(* IEC 61131-3 sources: Std_PalletMover/Class/HAL_BMS_Base, 1 file *)

(* ---- HAL_BMS_Base.st ---- *)
#define COMM_TIMEOUT              1000    // ms before timeout
#define TIMEOUTDELAY              15000    // Delay before checking for a communication timeout.

(*!
<Class
	Name               = "HAL_BMS_Base"
	Revision           = "0.0"
	RealtimeTask       = "false"
	CyclicTask         = "false"
	BackgroundTask     = "false"
	Sigmatek           = "false"
	OSInterface        = "false"
	HighPriority       = "false"
	Automatic          = "false"
	UpdateMode         = "Prescan"
	SharedCommandTable = "true"
	Objectsize         = "(284,120)">
	<Channels>
		<Server Name="ClassSvr" Visualized="false" Initialize="false" WriteProtected="true" Retentive="false"/>
	</Channels>
</Class>
*)
HAL_BMS_Base : CLASS
	TYPE
	  tBMSAlarms : BDINT  //! <Type Public="true" Name="tBMSAlarms"/>
	  [
	    1 ba_OverVoltage,
	    2 ba_UnderVoltage,
	    3 ba_AlmostUnderVoltage,
	    4 ba_BatteryEmpty,
	    5 ba_BatteryAlmostEmpty,
	    6 ba_InternalDefect,
	    7 ba_NoCommunication,
	    8 Bit8,
	    9 Bit9,
	    10 Bit10,
	    11 Bit11,
	    12 Bit12,
	    13 Bit13,
	    14 Bit14,
	    15 Bit15,
	    16 Bit16,
	    17 Bit17,
	    18 Bit18,
	    19 Bit19,
	    20 Bit20,
	    21 Bit21,
	    22 Bit22,
	    23 Bit23,
	    24 Bit24,
	    25 Bit25,
	    26 Bit26,
	    27 Bit27,
	    28 Bit28,
	    29 Bit29,
	    30 Bit30,
	    31 Bit31,
	    32 Bit32,
	  ];
#pragma pack(push, 1)
	  tBMSData : STRUCT  //! <Type Public="true" Name="tBMSData"/>
	    bd_StateOfCharge : UINT;
	    bd_TimeToGo : UINT;
	    bd_EnergyDraw : INT;
	    bd_BatteryVoltage : UINT;
	    bd_BatteryCurrent : INT;
	    bd_BatteryTemperature : INT;
	    bd_BatteryCharging : BOOL;
	    bd_BatteryLowIndication : BOOL;
	    bd_Alarm : tBMSAlarms;
	  END_STRUCT;
#pragma pack(pop)
	END_TYPE
  //Servers:
	ClassSvr 	: SvrChCmd_DINT;
  //Clients:
  //Variables:
  //Functions:

	FUNCTION VIRTUAL GLOBAL GetBMSData
		VAR_OUTPUT
			returnValue 	: tBMSData;
		END_VAR;
  //Tables:
	FUNCTION @STD
		VAR_OUTPUT
			ret_code	: CONFSTATES;
		END_VAR;
	FUNCTION GLOBAL TAB @CT_;
END_CLASS;

FUNCTION VIRTUAL GLOBAL HAL_BMS_Base::GetBMSData
  #pragma warning(disable: 73);
  #pragma warning(disable: 76);
	VAR_OUTPUT
		returnValue 	: tBMSData;
	END_VAR
  #pragma warning(default: 73);
  #pragma warning(default: 76);
END_FUNCTION
